// TIA Portal V21 export
VAR_GLOBAL   // PLC tag table "KAllAnalogica"
END_VAR
VAR_GLOBAL CONSTANT   // user constants
   KAllAnalog_Maxi : Int := 1;   // Maximale Schwelle ausgelöst / Maximum threshold reached / Umbral máximo intervenido / Seuil maximum intervenu / Soglia massima intervenuta
   KAllAnalog_IntMax : Int := 2;   // Maximale Zwischenschwelle ausgelöst / Maximum intermediate threshold intervened / Umbral intermedio máximo intervenido / Seuil intermédiaire maximal intervenu / Soglia intermedia massima intervenuta
   KAllAnalog_IntMin : Int := 3;   // Eingriffsminimaler Zwischenschwellenwert / Minimum intermediate threshold intervened / Umbral intermedio mínimo intervenido / Seuil intermédiaire minimal intervenu / Soglia intermedia minima intervenuta
   KAllAnalog_Mini : Int := 4;   // Eingriffsmindestschwelle / Minimum threshold intervened / Umbral mínimo intervenido / Seuil minimum intervenu / Soglia minima intervenuta
   KAllAnalog_OutOfRange : Int := 5;   // Sonde außerhalb des Messbereichs / Out of range of measurement / Sonda fuera del rango de medición / Sonde en dehors de la plage de mesure / Sonda fuori dal range di misurazione
END_VAR
